SUBAPPLICATION Softkey_Aux_Web_IE (* SoftKey ODER AUX (Joystick) ODER Web-Remote (extern zugefuehrter BOOL-Pegel, per AX_R_TRIG auf Flanke gewandelt) aktiviert -> 1 gemeinsames IND-Event. Baut auf Softkey_Aux_IE auf (Touchscreen+Joystick, diskreter Event-Kanal) und merged zusaetzlich den Web-Kanal hinzu - Muster fuer 'egal von welcher Quelle aus aktiviert, 1 Ergebnis-Event', z.B. Override-Erkennung. *)
  (* Standard: 61499-2 *)
  (* Version 2.0, 2026-09-16, Franz Höpfinger, ID-Parameter + internen SUBSCRIBE_R_TRIG (eigener lokaler OPC-UA-Self-Subscribe) entfernt, durch Socket WEB_IN (AX, Pegel von aussen) + AX_R_TRIG ersetzt - behebt Doppel-Self-Subscribe (FORTE: 'Cannot add another one'), da der Web-Knoten bereits von der Kommando-Seite (Softkey_Aux_Auto_IXA_TO_Remote_WRITE.WEB_STATE) abonniert wird. Siehe BERICHT_2026-09-16_STG3_I1_I3_I4_I6_STALE_REMOTE_SUBSCRIBE.md Abschnitt 16-17. *)
  (* Version 1.0, 2026-09-11, Franz Höpfinger, initial implementation *)
  PACKAGE MyLib::sys;
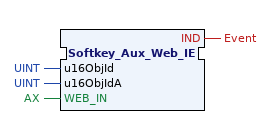
  EVENT_OUTPUT
    IND; (* Feuert wenn SoftKey ODER Aux ODER Web-Remote aktiviert wird *)
  END_EVENT
  VAR_INPUT
    u16ObjId : UINT; (* Object ID SoftKey *)
    u16ObjIdA : UINT; (* Object ID AuxFunction2 *)
  END_VAR
  SOCKETS
    WEB_IN : adapter::types::unidirectional::AX; (* Web-Remote-Pegel von aussen (z.B. Softkey_Aux_Auto_IXA_TO_Remote_WRITE.WEB_STATE), statt eigenem lokalen OPC-UA-Self-Subscribe *)
  END_SOCKETS
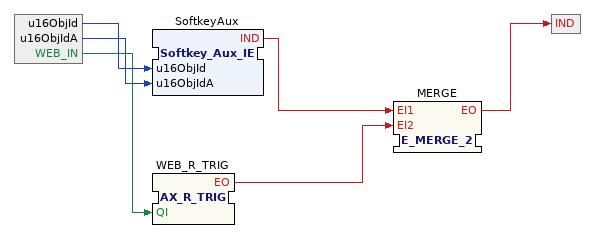
  FBS
    WEB_R_TRIG : adapter::events::unidirectional::AX_R_TRIG;
    MERGE : iec61499::events::E_MERGE_2;
  END_FBS
  SUBAPPS
    SoftkeyAux : MyLib::sys::Softkey_Aux_IE;
  END_SUBAPPS
  EVENT_CONNECTIONS
    SoftkeyAux.IND TO MERGE.EI1;
    WEB_R_TRIG.EO TO MERGE.EI2;
    MERGE.EO TO IND;
  END_CONNECTIONS
  DATA_CONNECTIONS
    u16ObjId TO SoftkeyAux.u16ObjId;
    u16ObjIdA TO SoftkeyAux.u16ObjIdA;
  END_CONNECTIONS
  ADAPTER_CONNECTIONS
    WEB_IN TO WEB_R_TRIG.QI;
  END_CONNECTIONS
END_SUBAPPLICATION
